// TwinCAT 3 PLC project Untitled1
// ProgramVersion: 3.1.4023.0
// libraries:
//   Tc2_Standard, * (Beckhoff Automation GmbH)
//   Tc2_System, * (Beckhoff Automation GmbH)
//   Tc3_Module, * (Beckhoff Automation GmbH)
//   VisuSymbols,3.5.10.0,System
// project tree:
//   / GlobalTextList.TcGTLO, PlcTask.TcTTO, 视图管理器.TcVMO (not stored)
//   POUs/ Convert.TcPOU, MAIN.TcPOU, TrafficLgiht.TcPOU
//   VISUs/ Visualization.TcVIS
// real-time tasks:
//   TASK PlcTask: cycle T#10ms, priority 20, ADS port 350

CONFIGURATION Untitled1
    RESOURCE PLC ON TwinCAT3
        TASK PlcTask(INTERVAL := T#10ms, PRIORITY := 20);
        PROGRAM MAIN WITH PlcTask : MAIN;
    END_RESOURCE
END_CONFIGURATION

// ---- POUs/MAIN.TcPOU
PROGRAM MAIN
VAR
;
END_VAR

TrafficLgiht();
Convert();

END_PROGRAM

// ---- POUs/TrafficLgiht.TcPOU
PROGRAM TrafficLgiht
VAR
	bStart:BOOL:=FALSE;
	Timer:TON;
	bNorthGreenLight:BOOL;
	bNorthYellowLight:BOOL;
	bNorthRedLight:BOOL;
	bWestGreenLight:BOOL;
	bWestYellowLight:BOOL;
	bWestRedLight:BOOL;
END_VAR

Timer(in:=NOT bStart ,PT:=T#20S);
bStart:=Timer.Q;

// Pass Between North South, not pass between West east
IF Convert.Timer>0 AND Convert.Timer<7000 THEN
	bNorthGreenLight:=1;
	bNorthYellowLight:=0;
	bNorthRedLight:=0;
	bWestGreenLight:=0;
	bWestYellowLight:=0;
	bWestRedLight:=1;
END_IF

// Wait Between North South, not pass between West east
IF Convert.Timer>7000 AND Convert.Timer<10000 THEN
	bNorthGreenLight:=0;
	bNorthYellowLight:=1;
	bNorthRedLight:=0;
	bWestGreenLight:=0;
	bWestYellowLight:=0;
	bWestRedLight:=1;
END_IF

// Not Pass Between North South , pass between West east
IF Convert.Timer>10000 AND Convert.Timer<17000 THEN
	bNorthGreenLight:=0;
	bNorthYellowLight:=0;
	bNorthRedLight:=1;
	bWestGreenLight:=1;
	bWestYellowLight:=0;
	bWestRedLight:=0;
END_IF

//  not pass Between North South, Wait between West east
IF Convert.Timer>17000 AND Convert.Timer<20000 THEN
	bNorthGreenLight:=0;
	bNorthYellowLight:=0;
	bNorthRedLight:=1;
	bWestGreenLight:=0;
	bWestYellowLight:=1;
	bWestRedLight:=0;
END_IF

END_PROGRAM

// ---- POUs/Convert.TcPOU
PROGRAM Convert
VAR
	Timer:INT;
END_VAR

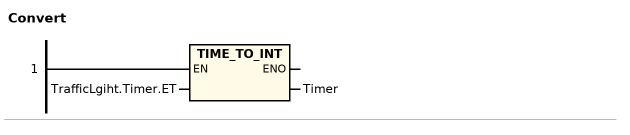
// NETWORK 1
Timer := TIME_TO_INT(TrafficLgiht.Timer.ET);

END_PROGRAM

// ---- VISUs/Visualization.TcVIS
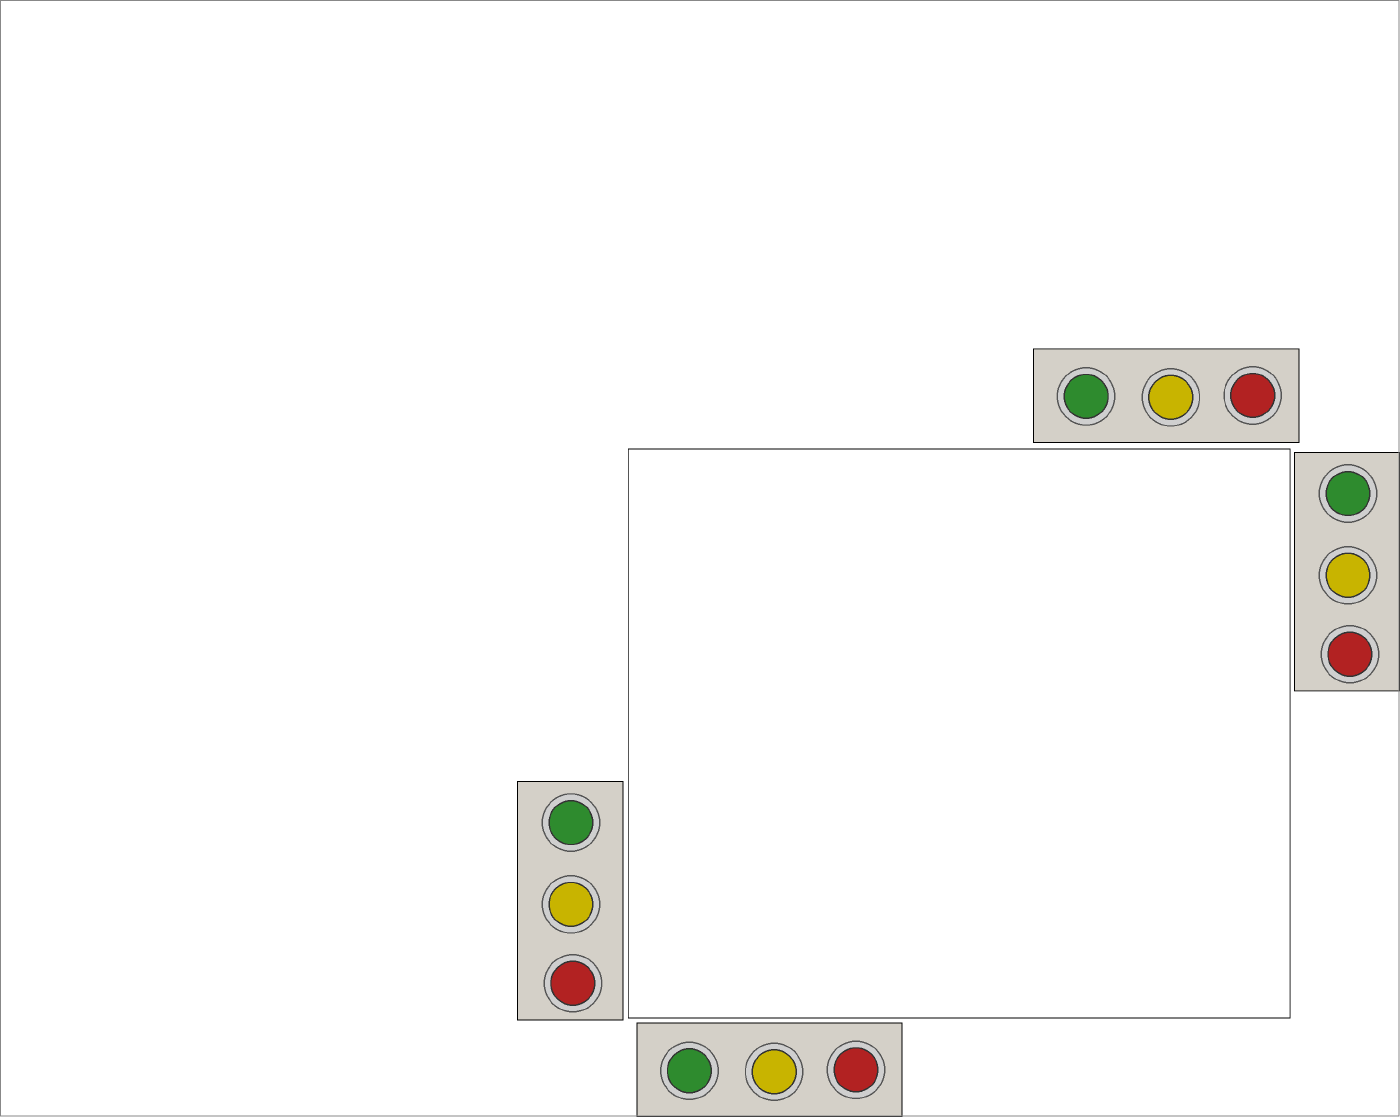
VISUALIZATION Visualization  // 1454x1161
    Group (1073,362 276x98)
        Rectangle (0,0 276x98)
        Lamp1 (20,15 70x70), variable: TrafficLgiht.bNorthGreenLight, style: Lamp-Lamp1-Green
        Lamp1 (193,14 70x70), variable: TrafficLgiht.bNorthRedLight, style: Lamp-Lamp1-Red
        Lamp1 (108,16 70x70), variable: TrafficLgiht.bNorthYellowLight, style: Lamp-Lamp1-Yellow
    Group (537,812 110x248)
        Rectangle (0,0 110x248)
        Lamp1 (21,8 70x70), variable: TrafficLgiht.bWestGreenLight, style: Lamp-Lamp1-Green
        Lamp1 (23,175 70x70), variable: TrafficLgiht.bWestRedLight, style: Lamp-Lamp1-Red
        Lamp1 (21,93 70x70), variable: TrafficLgiht.bWestYellowLight, style: Lamp-Lamp1-Yellow
    Rectangle (652,466 688x592)
    Group (661,1063 276x98)
        Rectangle (0,0 276x98)
        Lamp1 (20,15 70x70), variable: TrafficLgiht.bNorthGreenLight, style: Lamp-Lamp1-Green
        Lamp1 (193,14 70x70), variable: TrafficLgiht.bNorthRedLight, style: Lamp-Lamp1-Red
        Lamp1 (108,16 70x70), variable: TrafficLgiht.bNorthYellowLight, style: Lamp-Lamp1-Yellow
    Group (1344,470 110x248)
        Rectangle (0,0 110x248)
        Lamp1 (21,8 70x70), variable: TrafficLgiht.bWestGreenLight, style: Lamp-Lamp1-Green
        Lamp1 (23,175 70x70), variable: TrafficLgiht.bWestRedLight, style: Lamp-Lamp1-Red
        Lamp1 (21,93 70x70), variable: TrafficLgiht.bWestYellowLight, style: Lamp-Lamp1-Yellow
END_VISUALIZATION
